(* CODESYS project IndraLogic.project

Project tree, tasks and I/O mapping:
  MLD : IndraDrive MLD-2G MPx20, Bosch Rexroth AG, order no. FWA-INDRV_-MPx-20VRS, version 20.24.1422.3503
    application Application
      libraries: Linked List, 1.2.1.14 (Bosch Rexroth); MQTT Client, 2.3.8.14 (Bosch Rexroth)
      task PlcTask (cyclic, interval t#20ms, priority 1) calls PlcProg
      global variables IO
      program PlcProg [ST]
    Parameter_IO : Drive I/O, Bosch Rexroth AG, version 20.1.2.0
        unmapped channels: Input P-0-1390, Input P-0-1391, Input P-0-1392, Input P-0-1393, Input P-0-1394, Input P-0-1395, Input P-0-1396, Input P-0-1397, Input P-0-1398, Input P-0-1399, Input P-0-1400, Input P-0-1401, Input P-0-1402, Input P-0-1403, Input P-0-1404, Input P-0-1405, Input P-0-1406, Input P-0-1407, Input P-0-1408, Input P-0-1409, Not Available, Not Available, Not Available, Not Available, Not Available, Not Available, Not Available, Not Available, Not Available, Not Available, Not Available, Not Available, Not Available, Not Available, Not Available, Input P-0-1440, Input P-0-1441, Input P-0-1442, Input P-0-1443, Input P-0-1444,
          Input P-0-1445, Input P-0-1446, Input P-0-1447, Output P-0-1410, Output P-0-1411, Output P-0-1412, Output P-0-1413, Output P-0-1414, Output P-0-1415, Output P-0-1416, Output P-0-1417, Output P-0-1418, Output P-0-1419, Output P-0-1420, Output P-0-1421, Output P-0-1422, Output P-0-1423, Output P-0-1424, Output P-0-1425, Output P-0-1426, Output P-0-1427, Output P-0-1428, Output P-0-1429
*)

// MLD/Application/IO
{attribute 'qualified_only'}
VAR_GLOBAL
	bEnableAxis AT %IX1.0 :BOOL;
	bExecuteVelocity AT %IX1.1 :BOOL;
	bChangeVelocity AT %IX1.2 :BOOL;
	bStopAxis AT %IX1.3 :BOOL;
END_VAR

// MLD/Application/PlcProg
PROGRAM PlcProg
VAR
	rVelocity 		: REAL;
	bIsAxisEnabled 	: BOOL;
	pwrOn			: MC_Power;
	moveVel			: MC_MoveVelocity;
	stopAxis		: MC_Stop;
	
END_VAR

VAR
	mqttClient 			: MQTTClientFB;
	mqttStatusPublish 	: MQTTPublishFB;
	mqttSubscribe 		: MQTTSubscribeFB;
	mqttString 			: MQTTGetStringFB;
	
	sMQTT_TOPIC_SERVO_CMD 	: STRING :='SERVO/CMD';
	sMQTT_TOPIC_CONNECTION 	: STRING :='SERVO/CONNECTION';
	
	sPayloads				: STRING:='Connected';
	
	sMES 			: STRING;
	sCMD 			: STRING;
	rVel			: REAL;
	
END_VAR

mqttClient(
	Enable:= TRUE, 
	IPAddress:='192.168.99.187', 
	Port:= , 
	ConnectionTimeout:= , 
	KeepAlive:= 10, 
	ClientID:= 'plcClient', 
	Username:= , 
	Password:= , 
	LastWillRetain:= TRUE, 
	LastWillTopic:= , 
	LastWillMessage:= 'OFFLINE', 
	LastWillQos:= , 
	TCPConnected=> , 
	Connected=> , 
	Socket=> , 
	PubAckID=> , 
	ErrorCode=> , 
	ErrorInfo=> , 
	ConnectionState=> , 
	SubscribedDataRecvd=> );
	
mqttSubscribe(
	Enable:= mqttClient.Connected, 
	Post:= , 
	Topic:= sMQTT_TOPIC_SERVO_CMD, 
	QoS:= ,  
	ConnectionHandle:= ADR(mqttClient), 
	ErrorCode=> , 
	RunningState=> , 
	Complete=> , 
	Retries=> );

		
mqttString(
	Enable:= mqttSubscribe.Complete, 
	Topic:= sMQTT_TOPIC_SERVO_CMD, 
	Prefix:= , 
	Enabled=> , 
	Output=> sMES, 
	Done=> );	
	
mqttStatusPublish(
	Enable:= mqttClient.Connected, 
	Post:= , 
	Retained:= , 
	QoS:= , 
	Topic:= sMQTT_TOPIC_CONNECTION , 
	Payload:= ADR(sPayloads), 
	DataLength:= INT_TO_UINT(len(sPayloads)) , 
	ConnectionHandle:= ADR(mqttClient) , 
	ErrorCode=> , 
	RunningState=> );

IF mqttString.Done THEN
	sCMD := LEFT(sMES,2);
	rVel := STRING_TO_REAL(DELETE(sMes,2,1));
	IF sMES = 'RUN' OR sMES = 'run' THEN
		pwrOn.Enable := TRUE;
		IF sCMD = 'RV' AND rVel > 0 AND rVel < 200 THEN
			rVelocity := rVel;
		ELSIF sCMD = 'LV' AND rVel > 0 AND rVel < 200 THEN
			rVelocity := -1 * rVel;
		END_IF
	ELSIF sMES = 'STOP' OR sMES = 'stop' THEN
		stopAxis.Execute := TRUE;
		pwrOn.Enable := FALSE;
	END_IF
END_IF


 
	
pwrOn(
	Enable:= ,
	Status=> bIsAxisEnabled, 
	Error=> , 
	ErrorID=> , 
	ErrorIdent=> , 
	Axis:= Axis3 );
	
moveVel(
	Execute:= , 
	Velocity:= rVelocity, 
	Acceleration:= 1000, 
	Deceleration:= 1000, 
	InVelocity=> , 
	Active=> , 
	CommandAborted=> , 
	Error=> , 
	ErrorID=> , 
	ErrorIdent=> , 
	Axis:= Axis3);
	
stopAxis(
	Execute:= , 
	Deceleration:= 1000, 
	Done=> , 
	Active=> , 
	CommandAborted=> , 
	Error=> , 
	ErrorID=> , 
	ErrorIdent=> , 
	Axis:= Axis3);

END_PROGRAM
